FUNCTION_BLOCK AGRIPPER_DEMUX (* Composite FB wrapping other FBs *)
  (* Standard: 61499-2 *)
  (* Version 0.0, 2008-07-10, 4DIAC-IDE, 4DIAC-Consortium *)
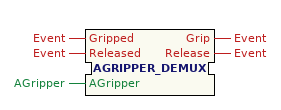
  EVENT_INPUT
    Gripped; (* Request from Socket *)
    Released; (* Response from Socket *)
  END_EVENT
  EVENT_OUTPUT
    Grip; (* Confirmation from Plug *)
    Release; (* Indication from Plug *)
  END_EVENT
  SOCKETS
    AGripper : AGripper;
  END_SOCKETS
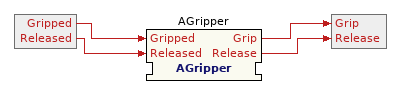
  EVENT_CONNECTIONS
    Gripped TO AGripper.Gripped;
    Released TO AGripper.Released;
    AGripper.Grip TO Grip;
    AGripper.Release TO Release;
  END_CONNECTIONS
END_FUNCTION_BLOCK
